// Precision: 100ns.
FUNCTION GetUnixTime : ULINT
VAR_INPUT
END_VAR
VAR
END_VAR

GetUnixTime := Tc2_System.F_GetSystemTime() - 11_644_473_678_000_000_0;

END_FUNCTION

(* stored: Version 1.1.0.1
   POU GetUnixTime: Id {9256dbe0-970c-46b2-beb0-50dc80b906e9}, SpecialFunc None *)
